SYSTEM Simple Test System
  (* Version 1.0, 2008-01-17, Goran Cengic, Chalmers *)
  DEVICE Test Device : DeviceType_not_used
    RESOURCE Test Resource : ResourceType_not_used
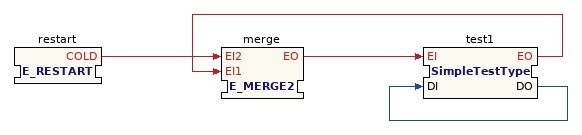
      FBS
        restart : E_RESTART;
        merge : E_MERGE2;
        test1 : SimpleTestType;
      END_FBS
      EVENT_CONNECTIONS
        restart.COLD TO merge.EI2;
        merge.EO TO test1.EI;
        test1.EO TO merge.EI1;
      END_CONNECTIONS
      DATA_CONNECTIONS
        test1.DO TO test1.DI;
      END_CONNECTIONS
    END_RESOURCE
  END_DEVICE
END_SYSTEM
